// TIA Portal project "260609_V003_DreiBänderAufgabeParameterFC" (V17)

(* hardware
DEVICE "S7-1500/ET200MP-Station_1"  S7-1500 station
   slot 0: "Profilschiene_0"  Rack  6ES7 590-1***0-0AA0
   slot 0: "PM 70W 120/230VAC"  PM 70W 120/230VAC  6EP1332-4BA00
   slot 1: "PLC_1"  CPU 1516-3 PN/DP  6ES7 516-3AN02-0AB0  V2.9
      slot 3: "CPU-Display_1"  6ES7591-1BA00-0AA0
      slot 32768: "PROFINET-Schnittstelle_1"  X1
         slot 32769: "Port_1"  X1 P1
         slot 32770: "Port_2"  X1 P2
      slot 33024: "PROFINET-Schnittstelle_2"  X2
         slot 33025: "Port_1"  X2 P1
      slot 33280: "DP-Schnittstelle_1"  X3
      slot 34817: "Virtual CP interface port_1"  Virtual CP interface port  Virtual CP interface port
   slot 2: "DI 32x24VDC HF_1"  DI 32x24VDC HF  6ES7 521-1BL00-0AB0  V2.1
   slot 3: "DQ 32x24VDC/0.5A ST_1"  DQ 32x24VDC/0.5A ST  6ES7 522-1BL00-0AB0  V2.0
   slot 4: "AI 8xU/I/RTD/TC ST_1"  AI 8xU/I/RTD/TC ST  6ES7 531-7KF00-0AB0  V2.2
   slot 5: "AQ 4xU/I ST_1"  AQ 4xU/I ST  6ES7 532-5HD00-0AB0  V2.1
   slot 6: "DI 16x24VDC BA_1"  DI 16x24VDC BA  6ES7 521-1BH10-0AA0  V1.1
   slot 7: "DI 16x24VDC HS_1"  DI 16x24VDC HS  6ES7 521-7BH00-0AB0  V1.0
   slot 8: "DI 16x24VDC HF_1"  DI 16x24VDC HF  6ES7 521-1BH00-0AB0  V2.2
*)

// ===== PLC "PLC_1"  CPU 1516-3 PN/DP =====

VAR_GLOBAL   // PLC tag table "Standard-Variablentabelle"
   "S0_Not-Aus" AT %E0.0 : Bool;
   "S1_Anlage ein" AT %E0.1 : Bool;
   "S2Bänder starten" AT %E0.2 : Bool;
   "S3Bänder stoppen" AT %E0.3 : Bool;
   "S4Reset Not-Aus" AT %E0.4 : Bool;
   "F5_MSS_Motor1" AT %E0.5 : Bool;
   "F7_MSS_Motor2" AT %E0.6 : Bool;
   "F9_MSS_Motor3" AT %E0.7 : Bool;
   "FRG_Motor" AT %M10.0 : Bool;
   "AnlageEIN" AT %M10.1 : Bool;
   "BänderEIN" AT %M10.2 : Bool;
   "Q1_Motor1" AT %A0.0 : Bool;   // Ansteuerung Motor 1, Band1
   "SE_Q1Motor1" AT %T10 : Timer;
   "SA_Q1Motor1" AT %T11 : Timer;
   "Q2_Motor2" AT %A0.1 : Bool;   // Ansteuerung Motor 2, Band2
   "Q3_Motor3" AT %A0.2 : Bool;   // Ansteuerung Motor 3, Band3
   "SE_Q2Motor2" AT %T12 : Timer;
   "SA_Q2Motor2" AT %T13 : Timer;
   "SE_Q3Motor3" AT %T14 : Timer;
   "SA_Q3Motor3" AT %T15 : Timer;
   "B1_BehälterVorhanden" AT %E1.0 : Bool;
   "B2_BehälterVorhanden" AT %E1.1 : Bool;
   "P1_MSS_OK" AT %A0.3 : Bool;
END_VAR

FUNCTION "fc002_FreigabeMotore" : Void   // FC2, FBD
{ S7_Optimized_Access := 'TRUE' }
VERSION : 0.1
   VAR_TEMP
      MSS_OK : Bool;
   END_VAR
BEGIN

REGION Network 1
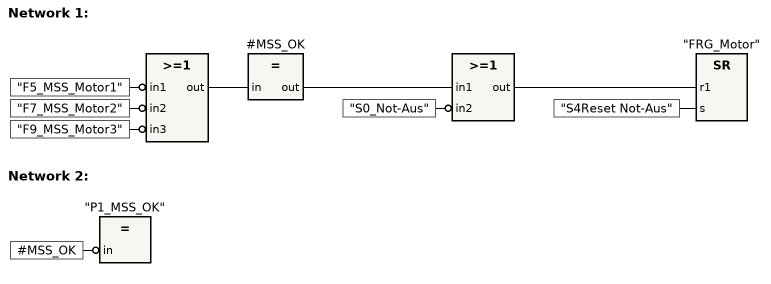
   #MSS_OK := NOT "F5_MSS_Motor1" OR NOT "F7_MSS_Motor2" OR NOT "F9_MSS_Motor3";
   IF "S4Reset Not-Aus" THEN
       "FRG_Motor" := TRUE;   // SR flip-flop
   END_IF;
   IF #MSS_OK OR NOT "S0_Not-Aus" THEN "FRG_Motor" := FALSE; END_IF;
END_REGION

REGION Network 2
   "P1_MSS_OK" := NOT #MSS_OK;
END_REGION
END_FUNCTION

FUNCTION "fc003_Betriebsarten" : Void   // FC3, FBD
{ S7_Optimized_Access := 'TRUE' }
VERSION : 0.1
BEGIN

REGION Network 1: Betriebsart AnlageEIN
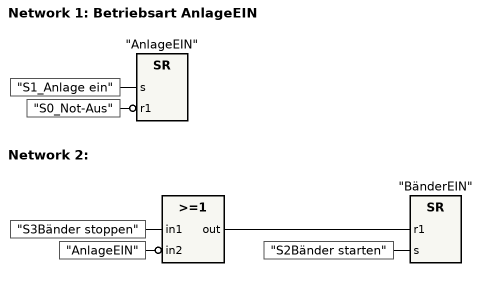
   IF "S1_Anlage ein" THEN
       "AnlageEIN" := TRUE;   // SR flip-flop
   END_IF;
   IF NOT "S0_Not-Aus" THEN "AnlageEIN" := FALSE; END_IF;
END_REGION

REGION Network 2
   IF "S2Bänder starten" THEN
       "BänderEIN" := TRUE;   // SR flip-flop
   END_IF;
   IF "S3Bänder stoppen" OR NOT "AnlageEIN" THEN "BänderEIN" := FALSE; END_IF;
END_REGION
END_FUNCTION

FUNCTION "fc010_AnsteuerungAntriebe" : Void   // FC10, FBD
{ S7_Optimized_Access := 'TRUE' }
VERSION : 0.1
   VAR_TEMP   // added for the SCL form of the ladder/FBD networks
      _w1 : Bool;
      _s5time1 : S5Time;
      _w2 : Bool;
      _s5time2 : S5Time;
   END_VAR
BEGIN

REGION Network 1: Ansteuerung Motor 1, Band1
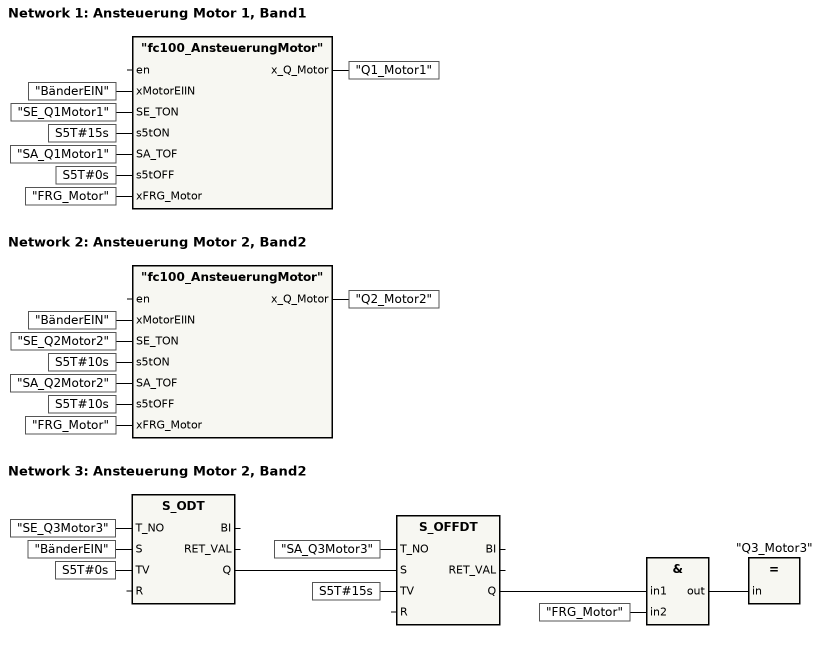
   "fc100_AnsteuerungMotor"(xMotorEIIN := "BänderEIN",
                           SE_TON := "SE_Q1Motor1",
                           s5tON := S5T#15s,
                           SA_TOF := "SA_Q1Motor1",
                           s5tOFF := S5T#0s,
                           xFRG_Motor := "FRG_Motor",
                           x_Q_Motor => "Q1_Motor1");
END_REGION

REGION Network 2: Ansteuerung Motor 2, Band2
   "fc100_AnsteuerungMotor"(xMotorEIIN := "BänderEIN",
                           SE_TON := "SE_Q2Motor2",
                           s5tON := S5T#10s,
                           SA_TOF := "SA_Q2Motor2",
                           s5tOFF := S5T#10s,
                           xFRG_Motor := "FRG_Motor",
                           x_Q_Motor => "Q2_Motor2");
END_REGION

REGION Network 3: Ansteuerung Motor 2, Band2
   #_s5time1 := S_ODT(T_NO := "SE_Q3Motor3", S := "BänderEIN", TV := S5T#0s, Q => #_w1);
   #_s5time2 := S_OFFDT(T_NO := "SA_Q3Motor3", S := #_w1, TV := S5T#15s, Q => #_w2);
   "Q3_Motor3" := #_w2 AND "FRG_Motor";
END_REGION
END_FUNCTION

FUNCTION "fc100_AnsteuerungMotor" : Void   // FC100, FBD
{ S7_Optimized_Access := 'TRUE' }
VERSION : 0.1
   VAR_INPUT
      xMotorEIIN : Bool;
      SE_TON : Timer;
      s5tON : S5Time;
      SA_TOF : Timer;
      s5tOFF : S5Time;
      xFRG_Motor : Bool;
   END_VAR
   VAR_OUTPUT
      x_Q_Motor : Bool;
   END_VAR
   VAR_TEMP   // added for the SCL form of the ladder/FBD networks
      _w1 : Bool;
      _s5time1 : S5Time;
      _w2 : Bool;
      _s5time2 : S5Time;
   END_VAR
BEGIN

REGION Network 1: Ansteuerung Motor 1, Band1
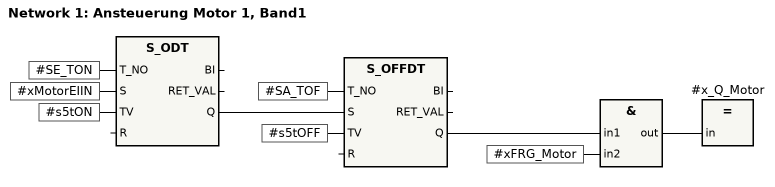
   #_s5time1 := S_ODT(T_NO := #SE_TON, S := #xMotorEIIN, TV := #s5tON, Q => #_w1);
   #_s5time2 := S_OFFDT(T_NO := #SA_TOF, S := #_w1, TV := #s5tOFF, Q => #_w2);
   #x_Q_Motor := #_w2 AND #xFRG_Motor;
END_REGION
END_FUNCTION

ORGANIZATION_BLOCK "Main"   // OB1, FBD, ProgramCycle
TITLE = "Main Program Sweep (Cycle)"
{ S7_Optimized_Access := 'TRUE' }
VERSION : 0.1
   VAR_INPUT
      Initial_Call : Bool;   // Initial call of this OB
      Remanence : Bool;   // =True, if remanent data are available
   END_VAR
BEGIN

REGION Network 1
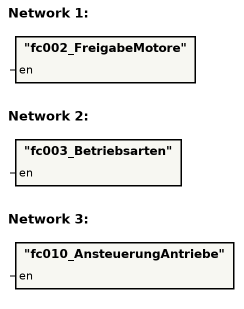
   "fc002_FreigabeMotore"();
END_REGION

REGION Network 2
   "fc003_Betriebsarten"();
END_REGION

REGION Network 3
   "fc010_AnsteuerungAntriebe"();
END_REGION
END_ORGANIZATION_BLOCK